# EPICS substitutions: ek9000App/Db/EL3202.substitutions
file EL3202.template
{       pattern
        {
                TERMINAL,

        }
        {
        }
}
